FUNCTION_BLOCK Test_TStreamAdd_Read_LREAL EXTENDS T_UnitTestBase
VAR
    Stream : T_Stream(StreamLength := 2);
END_VAR



Stream.Init(2);

Stream.Add_LREAL(1.234567891234);
    
Assertion.AssertEquals_UDINT(
    Expected := 10,
    Actual := Stream.Position,
    VariableName := 'Stream.Position');
    
Stream.Seek(0);

Assertion.AssertEquals_LREAL(
    Expected := 1.234567891234,
    Actual := Stream.Read_LREAL(),
    Delta  := 0.000000000001,
    VariableName := 'Stream.Read_LREAL()');
    
Assertion.AssertEquals_UDINT(
    Expected := 10,
    Actual := Stream.Position,
    VariableName := 'Stream.Position');
    
    
TestFinished();

END_FUNCTION_BLOCK

(* stored: Version 1.1.0.1, ProductVersion 3.1.4024.6
   POU Test_TStreamAdd_Read_LREAL: Id {ce91e671-6f43-49fd-900c-f9fba041ddbb}, SpecialFunc None *)
